FUNCTION_BLOCK ADD_1990CFD1468AAE4A6 (* Add *)
  (* Standard: 61499-2 *)
  (* Version 1.0, 24.09.2008, marumil, nxtControl GmbH, Initial Version *)
  PACKAGE Main;
  (* Compiler Cpp *)
  {SET_ATTRIBUTE(Runtime.FBType.ImplementingType, Runtime.Standard#DYNGEN_ADD)}
  {SET_ATTRIBUTE(Configuration.GenericFBType.InterfaceParams, Runtime.Standard#CNT:=2;IN${CNT$}:LREAL)}
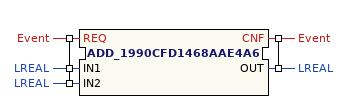
  EVENT_INPUT
    REQ WITH IN1, IN2; (* Normal Execution Request *)
  END_EVENT
  EVENT_OUTPUT
    CNF WITH OUT; (* Execution Confirmation *)
  END_EVENT
  VAR_INPUT
    IN1 : LREAL; (* Argument *)
    IN2 : LREAL; (* Argument *)
  END_VAR
  VAR_OUTPUT
    OUT : LREAL; (* Result: IN1 + IN2 + ... *)
  END_VAR
  EC_STATES
    START;
  END_STATES
END_FUNCTION_BLOCK
